SUBAPPLICATION Seitenschieber (* Subapplication Type *)
  (* Standard: 61499-2 *)
  (* Version 1.0, 2023-01-29, Franz *)
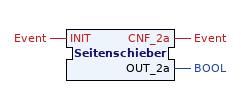
  EVENT_INPUT
    INIT;
  END_EVENT
  EVENT_OUTPUT
    CNF_2a;
  END_EVENT
  VAR_OUTPUT
    OUT_2a : BOOL;
  END_VAR
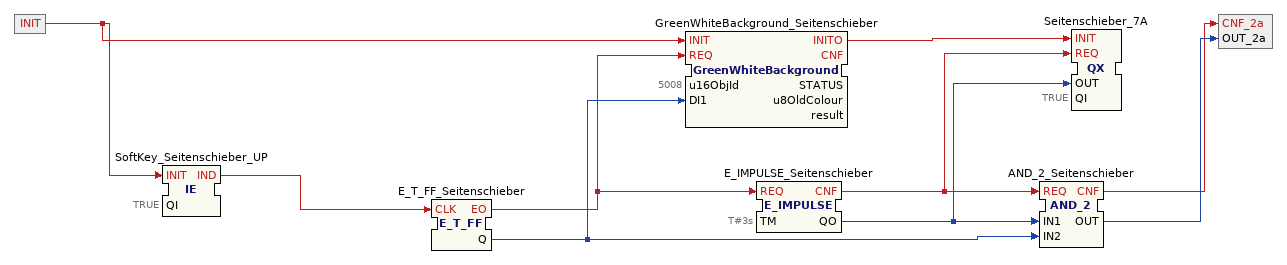
  FBS
    GreenWhiteBackground_Seitenschieber : GreenWhiteBackground(u16ObjId := 5008);
    E_IMPULSE_Seitenschieber : E_IMPULSE(TM := T#3s);
    AND_2_Seitenschieber : AND_2;
    E_T_FF_Seitenschieber : E_T_FF;
    Seitenschieber_7A : QX(QI := TRUE);
    SoftKey_Seitenschieber_UP : IE(QI := TRUE);
  END_FBS
  EVENT_CONNECTIONS
    E_T_FF_Seitenschieber.EO TO GreenWhiteBackground_Seitenschieber.REQ;
    GreenWhiteBackground_Seitenschieber.INITO TO Seitenschieber_7A.INIT;
    E_T_FF_Seitenschieber.EO TO E_IMPULSE_Seitenschieber.REQ;
    E_IMPULSE_Seitenschieber.CNF TO Seitenschieber_7A.REQ;
    E_IMPULSE_Seitenschieber.CNF TO AND_2_Seitenschieber.REQ;
    AND_2_Seitenschieber.CNF TO CNF_2a;
    INIT TO GreenWhiteBackground_Seitenschieber.INIT;
    INIT TO SoftKey_Seitenschieber_UP.INIT;
    SoftKey_Seitenschieber_UP.IND TO E_T_FF_Seitenschieber.CLK;
  END_CONNECTIONS
  DATA_CONNECTIONS
    E_T_FF_Seitenschieber.Q TO GreenWhiteBackground_Seitenschieber.DI1;
    E_IMPULSE_Seitenschieber.QO TO AND_2_Seitenschieber.IN1;
    E_IMPULSE_Seitenschieber.QO TO Seitenschieber_7A.OUT;
    E_T_FF_Seitenschieber.Q TO AND_2_Seitenschieber.IN2;
    AND_2_Seitenschieber.OUT TO OUT_2a;
  END_CONNECTIONS
END_SUBAPPLICATION
